# EPICS substitutions: ek9000App/Db/EL4134.substitutions
file EL4134.template
{       pattern
        {
                TERMINAL,

        }
        {
        }
}
